# EPICS autosave request: ADApp/Db/NDTimeSeriesN_settings.req
# This is for one signal
$(P)$(R)Name
$(P)$(R)Use
